(* IEC 61131-3 sources: generating_plc_code_with_llms/Code#1/ChatGPT_4/third run, 21 files *)

(* ---- 10.st ---- *)
//27.6s
//4
FUNCTION Sigmoid : REAL
VAR_INPUT
    x : REAL; // Input to the sigmoid function
END_VAR

// Sigmoid function calculation
Sigmoid := 1.0 / (1.0 + EXP(-x));

END_FUNCTION

(* ---- 11.st ---- *)
//22.62s
//4
FUNCTION Sign : INT
VAR_INPUT
    x : REAL; // Input to the sign function
END_VAR

// Determine the sign of the input x
IF x < 0 THEN
    Sign := -1; // x is negative
ELSIF x > 0 THEN
    Sign := 1; // x is positive
ELSE
    Sign := 0; // x is zero
END_IF

END_FUNCTION

(* ---- 12.st ---- *)
//30.77s
//4
FUNCTION HyperbolicSine : REAL
VAR_INPUT
    x : REAL; // Input to the hyperbolic sine function
END_VAR

// Hyperbolic sine calculation using the exponential function
HyperbolicSine := (EXP(x) - EXP(-x)) / 2.0;

END_FUNCTION

(* ---- 14.st ---- *)
// 39.74s
// 4
FUNCTION FC1001 : BOOL
VAR_INPUT
    MeasuredValue: REAL; // Sensor measured value
    SwitchingValue: REAL; // Predeterminable switching value
    HysteresisPct: REAL; // Hysteresis percentage
END_VAR

VAR
    HysteresisValue: REAL;
END_VAR

BEGIN
    // Calculate the hysteresis value
    HysteresisValue := (SwitchingValue * HysteresisPct) / 100.0;

    // Check if the measured value exceeds the switching value + hysteresis
    IF MeasuredValue > (SwitchingValue + HysteresisValue) THEN
        FC1001 := TRUE; // Turn on the output
    ELSIF MeasuredValue < (SwitchingValue - HysteresisValue) THEN
        FC1001 := FALSE; // Turn off the output
    END_IF;
END_FUNCTION

(* ---- 15.st ---- *)
// 49.09s
// 3
FUNCTION FC1002 : VOID
VAR_INPUT
    Detected: BOOL;    // Detection by ultrasonic sensor
    SystemOn: BOOL;    // System on/off switch (E_A)
END_VAR

VAR_OUTPUT
    P_HU: BOOL;        // Horn for acoustic warning
    P_AL: BOOL;        // Alarm signal
    P1: BOOL;          // System on indicator
END_VAR

VAR
    DetectionTimer: TON; // Timer for detection duration
END_VAR

BEGIN
    IF SystemOn THEN
        P1 := TRUE; // Indicate system is on

        IF Detected THEN
            IF NOT DetectionTimer.IN THEN
                DetectionTimer(IN := TRUE, PT := T#3s); // Start timer when object is detected
            END_IF;

            IF NOT DetectionTimer.Q THEN
                P_HU := TRUE; // Activate warning horn if object detected
            ELSE
                P_HU := FALSE;
                P_AL := TRUE; // Activate alarm if object detected for more than 3 seconds
            END_IF;
        ELSE
            DetectionTimer(IN := FALSE); // Reset timer if no object is detected
            P_HU := FALSE;
        END_IF;
    ELSE
        P1 := FALSE; // Indicate system is off
        DetectionTimer(IN := FALSE); // Reset timer
        P_HU := FALSE;
        P_AL := FALSE; // Reset alarm
    END_IF;
END_FUNCTION

(* ---- 18.st ---- *)
// 41.17s
// 2
FUNCTION FC1003 : REAL
VAR_INPUT
    InputValue: WORD; // The input value from the temperature sensor (0 to 255)
    IN_MIN, IN_MAX: WORD; // Input range lower and upper limits
    OUT_MIN, OUT_MAX: REAL; // Output range lower and upper limits
END_VAR

BEGIN
    // Linear interpolation
    FC1003 := OUT_MIN + ((REAL(InputValue) - REAL(IN_MIN)) * (OUT_MAX - OUT_MIN)) / (REAL(IN_MAX) - REAL(IN_MIN));
END_FUNCTION

(* ---- 3.st ---- *)
//25.24s
//2
FUNCTION Fibonacci : DINT
VAR_INPUT
    n : DINT; // The nth Fibonacci number to calculate
END_VAR
VAR
    a : DINT := 0;
    b : DINT := 1;
    i : DINT;
    temp : DINT;
END_VAR

// Handle the base cases
IF n = 0 THEN
    RETURN 0;
ELSIF n = 1 THEN
    RETURN 1;
END_IF

// Calculate the nth Fibonacci number iteratively
FOR i := 2 TO n DO
    temp := a + b;
    a := b;
    b := temp;
END_FOR

RETURN b;
END_FUNCTION

(* ---- 8.st ---- *)
//32.73s
//2
FUNCTION LambertW : REAL
VAR_INPUT
    x : REAL; // Input value for which to compute W(x)
END_VAR
VAR
    w : REAL := 0; // Initial guess for W(x)
    tol : REAL := 1e-5; // Tolerance for stopping the iteration
    maxIter : INT := 100; // Maximum number of iterations
    iter : INT := 0; // Iteration counter
    diff : REAL; // Difference between successive iterations
END_VAR

// Check for the special case of x = 0
IF x = 0 THEN
    RETURN 0;
END_IF

// Check for a reasonable starting point for x > e or x < -1/e
IF x > 2.71828 OR x < -0.367879 THEN
    w := x;
ELSE
    w := LOG(x); // Start with natural logarithm of x for better convergence if x is within a typical range
END_IF

// Newton-Raphson iteration for the Lambert W function
REPEAT
    diff := (w * EXP(w) - x) / (EXP(w) + w * EXP(w));
    w := w - diff;
    iter := iter + 1;
UNTIL (ABS(diff) < tol) OR (iter >= maxIter);

// Check for non-convergence
IF iter >= maxIter THEN
    w := -1; // An error value to indicate non-convergence
END_IF

RETURN w;
END_FUNCTION

(* ---- 19.st ---- *)
// 62.53s
// 2
FUNCTION_BLOCK FB1005
VAR_INPUT
    START: BOOL;      // Sensor signal for measurement start/end
    THICKNESS: DWORD; // Thickness measurement from lasers
    V_MAX, V_MIN: REAL; // Tolerance band limits
END_VAR

VAR_OUTPUT
    M_MAX, M_MIN: DWORD; // Maximum and Minimum thickness measurements
    P1: BOOL;            // Reject light
END_VAR

VAR
    CurrentValue: REAL;
    MeasurementInProgress: BOOL := FALSE;
END_VAR

BEGIN
    IF START AND NOT MeasurementInProgress THEN
        // Start of a new measurement
        MeasurementInProgress := TRUE;
        M_MAX := 0;
        M_MIN := DWORD(MAX_INT); // Set to maximum possible value
    ELSIF NOT START AND MeasurementInProgress THEN
        // End of measurement
        MeasurementInProgress := FALSE;

        // Check if the thickness values are outside the tolerance band
        IF (M_MAX > REAL_TO_DWORD(V_MAX)) OR (M_MIN < REAL_TO_DWORD(V_MIN)) THEN
            P1 := TRUE; // Activate reject light
        ELSE
            P1 := FALSE;
        END_IF;
    END_IF;

    IF MeasurementInProgress THEN
        // Convert thickness to REAL for comparison
        CurrentValue := DWORD_TO_REAL(THICKNESS);

        // Update max and min values
        IF CurrentValue > DWORD_TO_REAL(M_MAX) THEN
            M_MAX := THICKNESS;
        END_IF;
        IF CurrentValue < DWORD_TO_REAL(M_MIN) THEN
            M_MIN := THICKNESS;
        END_IF;
    END_IF;
END_FUNCTION_BLOCK

(* ---- 2.st ---- *)
//27.38s
//2
FUNCTION_BLOCK BinomialCoefficient
VAR_INPUT
    n : INT; // Total number of items
    k : INT; // Number of items to choose
END_VAR

VAR_OUTPUT
    result : LREAL; // The binomial coefficient result (using LREAL due to potential for large numbers)
END_VAR

VAR
    i : INT;
    numerator : LREAL := 1;
    denominator : LREAL := 1;
END_VAR

// Calculate the factorial for a given number
FUNCTION Factorial : LREAL
    VAR_INPUT
        value : INT;
    END_VAR
    VAR
        i : INT;
        fact : LREAL := 1;
    END_VAR
    FOR i := 2 TO value DO
        fact := fact * i;
    END_FOR
    Factorial := fact;
END_FUNCTION

// Calculate the binomial coefficient C(n, k)
METHOD Calculate : LREAL
    // Check for valid input
    IF (n < 0) OR (k < 0) OR (k > n) THEN
        result := -1; // Return -1 for invalid input
        RETURN;
    END_IF

    // Calculate n! / (k!(n-k)!)
    numerator := Factorial(n);
    denominator := Factorial(k) * Factorial(n - k);
    result := numerator / denominator;
    RETURN result;
END_METHOD
END_FUNCTION_BLOCK

(* ---- 21.st ---- *)
// 117.54s
// 2
FUNCTION_BLOCK BURNER
VAR_INPUT
    IN: BOOL;                    // Start control input
    OVER_TEMP: BOOL;             // Boiler over temperature protection
    OIL_TEMP: BOOL;              // Oil temperature readiness
    STAGE2: BOOL;                // Control input for activating stage 2
    RST: BOOL;                   // Reset input for clearing faults and lockout
END_VAR

VAR_OUTPUT
    PRE_HEAT: BOOL;              // Fuel oil warming activation output
    FAIL: BOOL;                  // Failure indication output
    STATUS: INT;                 // Status and error code output
END_VAR

VAR
    Timer: TON;                  // Timer for managing time delays
    LockoutTimer: TON;           // Lockout timer
    CurrentStage: INT := 110;    // Current operational stage
    Lockout: BOOL := FALSE;      // Lockout flag
END_VAR

// Constants for timing and stages (these should be adjusted as per requirements)
VAR CONSTANT
    PRE_HEAT_TIME: TIME := T#30s;
    SAFETY_TIME: TIME := T#60s;
    STAGE2_DELAY: TIME := T#120s;
    LOCKOUT_TIME: TIME := T#300s;
    PRE_VENTILATION_TIME: TIME := T#15s;
    PRE_IGNITE_TIME: TIME := T#5s;
    POST_IGNITE_TIME: TIME := T#10s;
END_VAR

// Implementation of the burner logic
BEGIN
    // Handle lockout period after faults
    IF Lockout THEN
        IF LockoutTimer(IN := TRUE, PT := LOCKOUT_TIME) THEN
            Lockout := FALSE;
            LockoutTimer(IN := FALSE); // Stop lockout timer
        END_IF;
        EXIT; // Exit the execution to ensure no operation during lockout
    END_IF;

    IF RST AND NOT LockoutTimer.Q THEN
        // Reset logic to clear faults and prepare for a new start
        FAIL := FALSE;
        STATUS := 110; // Wait for Start signal
        Lockout := FALSE;
        PRE_HEAT := FALSE;
        CurrentStage := 110;
    END_IF;

    IF OVER_TEMP THEN
        // Handle over temperature error
        FAIL := TRUE;
        STATUS := 9; // Error code for over temperature
        Lockout := TRUE;
        LockoutTimer(IN := TRUE, PT := LOCKOUT_TIME); // Start lockout timer
        EXIT; // Stop all operations immediately
    END_IF;

    IF IN AND NOT Lockout THEN
        // Start sequence and operational logic
        CASE CurrentStage OF
            110: // Standby, waiting for start signal
                IF IN THEN
                    PRE_HEAT := TRUE;
                    Timer(IN := TRUE, PT := PRE_HEAT_TIME);
                    CurrentStage := 111; // Startup sequence
                END_IF;
            111: // Startup sequence, waiting for OIL_TEMP signal
                IF OIL_TEMP THEN
                    Timer(IN := FALSE); // Stop the pre-heat timer
                    // Transition to next stage would be here, implementing further logic for fan, ignition, etc.
                    // This is a simplified representation
                    CurrentStage := 112; // Burner runs on stage 1
                ELSIF Timer.Q THEN
                    // Pre-heat time exceeded without reaching OIL_TEMP
                    FAIL := TRUE;
                    STATUS := 1; // Error code for pre-heat failure
                    Lockout := TRUE;
                    LockoutTimer(IN := TRUE, PT := LOCKOUT_TIME); // Start lockout timer
                END_IF;
            // Additional stages for fan operation, ignition, stage 2, etc., should be implemented here
        END_CASE;
    END_IF;
END_FUNCTION_BLOCK

(* ---- 1.st ---- *)
//18.66s
//4
PROGRAM AlarmControl
    VAR
        xAlarm1 : BOOL; // Alarm 1
        xAlarm2 : BOOL; // Alarm 2
        xAllOn  : BOOL; // Signal to turn all alarms on
        xAllOff : BOOL; // Signal to turn all alarms off
    END_VAR

    // Turn on both alarms if xAllOn is activated
    IF xAllOn THEN
        xAlarm1 := TRUE;
        xAlarm2 := TRUE;
        xAllOn := FALSE; // Reset the signal
    END_IF

    // Turn off both alarms if xAllOff is activated
    IF xAllOff THEN
        xAlarm1 := FALSE;
        xAlarm2 := FALSE;
        xAllOff := FALSE; // Reset the signal
    END_IF
END_PROGRAM

(* ---- 13.st ---- *)
//35.67s
//2
PROGRAM SearchNumber
VAR
    NumberList : ARRAY[1..100] OF INT; // List of random numbers
    i : INT := 1; // Loop counter starts at 1
    Found : BOOL := FALSE; // Flag to indicate if the number is found
    NumberToFind : INT := 10; // Number to find in the list
END_VAR

// Populate NumberList with random numbers for this example
// In a real-world scenario, this list would be populated differently
NumberList := [23, 56, 4, 67, 10, 1, 45, ... , 89]; // Continue filling the array with random numbers

// Search for the specific number
REPEAT
    IF NumberList[i] = NumberToFind THEN
        Found := TRUE;
        EXIT; // Exit the loop if the number is found
    END_IF

    i := i + 1;
UNTIL i > 100 OR Found;

// After the loop, check if the number was found
IF Found THEN
    // Code to handle the number found case
    // ...
ELSE
    // Code to handle the number not found case
    // ...
END_IF

END_PROGRAM

(* ---- 16.st ---- *)
//42.76s
//2
PROGRAM TrafficLightControl
VAR
    // Traffic Light Outputs
    North_green, North_yellow, North_red : BOOL;
    East_green, East_yellow, East_red : BOOL;

    // Timer
    CycleTimer : TON;

    // Constants for timing intervals
    CONST
        CYCLE_TIME : TIME := T#10000ms;
        NORTH_GREEN_TIME : TIME := T#5000ms;
        NORTH_YELLOW_TIME : TIME := T#500ms;
        EAST_GREEN_TIME : TIME := T#4000ms;
        EAST_YELLOW_TIME : TIME := T#500ms;
    END_CONST
END_VAR

CycleTimer(IN := TRUE, PT := CYCLE_TIME); // Timer is always running

// North light control
IF CycleTimer.ET < NORTH_GREEN_TIME THEN
    North_green := TRUE;
    North_yellow := FALSE;
    North_red := FALSE;
ELSIF CycleTimer.ET < (NORTH_GREEN_TIME + NORTH_YELLOW_TIME) THEN
    North_green := FALSE;
    North_yellow := TRUE;
    North_red := FALSE;
ELSE
    North_green := FALSE;
    North_yellow := FALSE;
    North_red := TRUE;
END_IF

// East light control
IF CycleTimer.ET >= NORTH_GREEN_TIME AND CycleTimer.ET < (NORTH_GREEN_TIME + NORTH_YELLOW_TIME) THEN
    East_green := FALSE;
    East_yellow := FALSE;
    East_red := TRUE;
ELSIF CycleTimer.ET >= (NORTH_GREEN_TIME + NORTH_YELLOW_TIME) AND CycleTimer.ET < (NORTH_GREEN_TIME + NORTH_YELLOW_TIME + EAST_GREEN_TIME) THEN
    East_green := TRUE;
    East_yellow := FALSE;
    East_red := FALSE;
ELSIF CycleTimer.ET >= (CYCLE_TIME - EAST_YELLOW_TIME) THEN
    East_green := FALSE;
    East_yellow := TRUE;
    East_red := FALSE;
ELSE
    East_green := FALSE;
    East_yellow := FALSE;
    East_red := TRUE;
END_IF

// Reset the timer if the cycle is complete
IF CycleTimer.ET >= CYCLE_TIME THEN
    CycleTimer(IN := FALSE); // Reset timer
    CycleTimer(IN := TRUE);  // Restart timer
END_IF
END_PROGRAM

(* ---- 17.st ---- *)
//41.87s
//2
PROGRAM WeatherStation
VAR
    nAnalogTempValue : INT; // Analog value from the temperature sensor
    nAnalogHumidValue : INT; // Analog value from the humidity sensor
    fTemperature : REAL; // Temperature in degrees Celsius
    fHumidity : REAL; // Humidity in percent
    sDisplayText : STRING; // Text to display in the house
END_VAR

// Constants for conversion (Assuming linear conversion, adjust as per your sensor specifications)
CONST
    TEMP_MIN : REAL := 0.0; // Minimum temperature sensor reading corresponds to
    TEMP_MAX : REAL := 50.0; // Maximum temperature sensor reading corresponds to
    HUMID_MIN : REAL := 0.0; // Minimum humidity sensor reading corresponds to
    HUMID_MAX : REAL := 100.0; // Maximum humidity sensor reading corresponds to
    ANALOG_MIN : INT := 0; // Minimum analog value
    ANALOG_MAX : INT := 32767; // Maximum analog value
END_CONST

// Convert the analog values to meaningful units
fTemperature := (fTemperature - TEMP_MIN) / (ANALOG_MAX - ANALOG_MIN) * (TEMP_MAX - TEMP_MIN);
fHumidity := (fHumidity - HUMID_MIN) / (ANALOG_MAX - ANALOG_MIN) * (HUMID_MAX - HUMID_MIN);

// Determine the temperature status
IF fTemperature < 18 THEN
    sDisplayText := 'Cold';
ELSIF fTemperature > 25 THEN
    sDisplayText := 'Hot';
ELSE
    // Nested IF for humidity check when temperature is between 18°C and 25°C
    IF fHumidity >= 40 AND fHumidity <= 75 THEN
        sDisplayText := 'Opt';
    ELSE
        sDisplayText := 'Temp. OK';
    END_IF
END_IF

END_PROGRAM

(* ---- 20.st ---- *)
// 36.75s
// 4
PROGRAM InterlockProgram
VAR
    I1, I2: BOOL;       // Inputs
    Q1, Q2: BOOL;       // Outputs
    TL: TIME;           // Dead time
    Timer1, Timer2: TON; // Timers for dead time
END_VAR

BEGIN
    // Timer logic for Q1
    IF NOT I2 AND (Timer2.Q OR NOT Timer2.IN) THEN
        IF I1 THEN
            Timer1(IN := TRUE, PT := TL);
            IF Timer1.Q THEN
                Q1 := TRUE;
            END_IF;
        ELSE
            Timer1(IN := FALSE);
            Q1 := FALSE;
        END_IF;
    ELSE
        Q1 := FALSE;
    END_IF;

    // Timer logic for Q2
    IF NOT I1 AND (Timer1.Q OR NOT Timer1.IN) THEN
        IF I2 THEN
            Timer2(IN := TRUE, PT := TL);
            IF Timer2.Q THEN
                Q2 := TRUE;
            END_IF;
        ELSE
            Timer2(IN := FALSE);
            Q2 := FALSE;
        END_IF;
    ELSE
        Q2 := FALSE;
    END_IF;
END_PROGRAM

(* ---- 4.st ---- *)
//36.02s
//2
PROGRAM FillLevelCheck
VAR
    nAnalogValue : INT; // Analog value input (0 - 32767)
    fFillLevel : REAL; // Converted fill level (0 - 100%)
    xLow : BOOL; // Output for low level
    xOk : BOOL; // Output for ok level
    xHigh : BOOL; // Output for high level
    xWarningHorn : BOOL; // Output for warning horn (<1%)
END_VAR

// Convert the analog value to a percentage
fFillLevel := REAL(nAnalogValue) * 100.0 / 32767.0;

// Check the fill level and set the outputs accordingly
CASE fFillLevel OF
    0.0 ..< 1.0:
        xLow := FALSE;
        xOk := FALSE;
        xHigh := FALSE;
        xWarningHorn := TRUE; // Activate warning horn if below 1%
    1.0 ..< 20.0:
        xLow := TRUE;
        xOk := FALSE;
        xHigh := FALSE;
        xWarningHorn := FALSE;
    20.0 ..< 80.0:
        xLow := FALSE;
        xOk := TRUE;
        xHigh := FALSE;
        xWarningHorn := FALSE;
    80.0 .. 100.0:
        xLow := FALSE;
        xOk := FALSE;
        xHigh := TRUE;
        xWarningHorn := FALSE;
    ELSE
        // Handle out of range values, if necessary
END_CASE

END_PROGRAM

(* ---- 5.st ---- *)
//35.75s
//4
PROGRAM GateController
VAR
    Start_Loop : BOOL; // Control variable to start the loop
    One_Hour_Timer : TON; // Timer that times out after 1 hour
    Gate_Is_Open : BOOL; // Indicates if the gate is open
    Sense_Car_App : BOOL; // Input that senses the car or the app
    Auth_String : STRING; // Authentication string provided by the car or app
    my_defined_str : STRING := 'YourAuthString'; // Predefined correct authentication string
    Timer_Done : BOOL; // Flag to indicate that the timer is done
END_VAR

// Check if the loop should start
IF NOT Start_Loop THEN
    IF NOT One_Hour_Timer.Q THEN // If the timer is not already done
        One_Hour_Timer(IN := TRUE, PT := T#1H); // Start or continue timing
    ELSE
        Timer_Done := TRUE; // Set the flag when the timer is done
    END_IF
ELSE
    One_Hour_Timer(IN := FALSE, PT := T#1H); // Reset the timer if Start_Loop is TRUE
    Timer_Done := FALSE; // Reset the flag
END_IF

// Timer logic to close the gate if it's still open after 1 hour
IF Timer_Done AND Gate_Is_Open THEN
    Gate_Is_Open := FALSE; // Close the gate
END_IF

// Logic to open the gate if the car or app is sensed and the authentication string matches
IF Sense_Car_App AND (Auth_String = my_defined_str) THEN
    Gate_Is_Open := TRUE; // Open the gate
END_IF

END_PROGRAM

(* ---- 6.st ---- *)
//49.52s
// 3
PROGRAM CraneLiftController
VAR
    // Inputs
    diConvTop : BOOL; // Top conveyor light barrier
    diConvBottom : BOOL; // Bottom conveyor light barrier
    diLiftTop : BOOL; // Lift at top position
    diLiftBottom : BOOL; // Lift at bottom position
    diLiftUnload : BOOL; // Lift at unloading position
    diBoxLift : BOOL; // Crate fully at the lift

    // Outputs
    doConvTop : BOOL; // Top conveyor belt control
    doConvBottom : BOOL; // Bottom conveyor belt control
    doConvLift : BOOL; // Lift conveyor belt control
    doLiftTop : BOOL; // Control to move lift to top
    doLiftBottom : BOOL; // Control to move lift to bottom
    doLiftUnload : BOOL; // Control to move lift to unload

    // Internal variables
    bTopRequested : BOOL; // Flag indicating top request
    bBottomRequested : BOOL; // Flag indicating bottom request
    bLiftMoving : BOOL; // Flag indicating lift is moving
    bUnloadProcess : BOOL; // Flag indicating unloading process
END_VAR

// Initial conveyor belt control - always on until light barriers are triggered
doConvTop := NOT diConvTop;
doConvBottom := NOT diConvBottom;

// Detect crate at top and request lift
IF diConvTop AND NOT bLiftMoving THEN
    bTopRequested := TRUE;
    bLiftMoving := TRUE;
    doConvTop := FALSE; // Stop top conveyor belt
END_IF

// Detect crate at bottom and request lift
IF diConvBottom AND NOT bLiftMoving THEN
    bBottomRequested := TRUE;
    bLiftMoving := TRUE;
    doConvBottom := FALSE; // Stop bottom conveyor belt
END_IF

// Lift movement logic
IF bLiftMoving THEN
    IF bTopRequested THEN
        doLiftTop := TRUE;
        doLiftBottom := FALSE;
        doLiftUnload := FALSE;
        IF diLiftTop THEN // When lift reaches top
            doConvLift := NOT diBoxLift; // Turn on lift conveyor until box is fully on
            IF diBoxLift THEN // Box is fully at lift
                bTopRequested := FALSE;
                bLiftMoving := FALSE;
                doLiftUnload := TRUE; // Move to unloading position
                bUnloadProcess := TRUE;
            END_IF
        END_IF
    ELSIF bBottomRequested THEN
        doLiftTop := FALSE;
        doLiftBottom := TRUE;
        doLiftUnload := FALSE;
        IF diLiftBottom THEN // When lift reaches bottom
            doConvLift := NOT diBoxLift; // Turn on lift conveyor until box is fully on
            IF diBoxLift THEN // Box is fully at lift
                bBottomRequested := FALSE;
                bLiftMoving := FALSE;
                doLiftUnload := TRUE; // Move to unloading position
                bUnloadProcess := TRUE;
            END_IF
        END_IF
    END_IF
END_IF

// Unloading process
IF bUnloadProcess AND diLiftUnload THEN
    doConvLift := TRUE; // Turn on lift conveyor to unload
    IF NOT diBoxLift THEN // Box has left the lift
        bUnloadProcess := FALSE;
        doLiftTop := FALSE; // Reset lift movement controls
        doLiftBottom := FALSE;
        doLiftUnload := FALSE;
        doConvLift := FALSE; // Stop lift conveyor
    END_IF
END_IF

END_PROGRAM

(* ---- 7.st ---- *)
//27.0s
// 2
PROGRAM CraneLoadCalculation
    // Constants
    CONST
        NUM_RECEPTORS : INT := 5;
        MAX_ANALOG_VALUE : INT := 32767;
    END_CONST

    // Variable Declarations
    VAR
        aiLoadReceptors : ARRAY[1..NUM_RECEPTORS] OF INT; // Array of analog input values from load receptors
        nTotalLoad : INT; // Variable to hold the total load
        fAverageLoad : REAL; // Variable to hold the average load
    END_VAR

    // Initialize total load
    nTotalLoad := 0;

    // Calculate the total load using a FOR loop
    FOR i := 1 TO NUM_RECEPTORS DO
        nTotalLoad := nTotalLoad + aiLoadReceptors[i];
    END_FOR

    // Calculate the average load
    IF nTotalLoad > 0 THEN
        fAverageLoad := REAL(nTotalLoad) / NUM_RECEPTORS;
    ELSE
        fAverageLoad := 0.0;
    END_IF
END_PROGRAM

(* ---- 9.st ---- *)
//21.55s
//4
PROGRAM LeapYearCheck
VAR
    YEAR : INT; // Variable holding the year to check
    IsLeapYear : BOOL; // Boolean variable indicating if it's a leap year
END_VAR

// Calculate if YEAR is a leap year
IsLeapYear := (YEAR MOD 4 = 0) AND ((YEAR MOD 100 <> 0) OR (YEAR MOD 400 = 0));

END_PROGRAM
